Universal Robots PolyScope program: velocity-move.urp

Program velocity-move (installation=default directory=/programs createdIn=5.2.0.61336 lastSavedIn=5.4.0.76181 robotSerialNumber=20195500451)
Calibrated DH parameters: a=[0.00002, -0.231658, -0.317125, 0.000011, 0.000055, 0]; d=[0.162082, 123.190176, -180.284242, 57.22734, 0.099524, 0.09934]; alpha=[1.569304, 0.00289, 0.004025, 1.569925, -1.569026, 0]; deltaTheta=[0, 0.993923, 4.662183, 0.627072, 0.000001, 0]
Robot Program (runOnlyOnce=true)
  Timer (action=Start) variable(name=time_start)
  angles := get_actual_joint_positions()
  Loop Forever
    Script: speedj([0.1*sin(time_start),0,0,0,0,0],15,0.002)
    var_1 := get_actual_joint_positions()
  Script: speedj([0,0,0,0,0,0],20,0.08)
  Wait Sleep waitTime=2
  MoveJ speed 60 deg/s, acceleration 80 deg/s^2 (useActiveTCP=true) feature=Base
    Waypoint Waypoint_2: TCP in base x=-612.643 y=103.453 z=303.743 mm, rx=2.3871 ry=-1.1583 rz=-0.7242 rad; joints [-178.101, -111.585, -105.31, -15.839, 95.595, 145.605] deg; TCP offset x=0 y=0 z=0 mm, rx=0 ry=0 rz=0 rad
    Halt
